// TIA Portal V16 export
// export: Created 2020-03-07T16:06:13.8131431Z, ExportSetting WithDefaults, DisplayName Totally Integrated Automation Portal, DisplayVersion V16 Update 1, DisplayName TIA Portal Version Control Interface, DisplayVersion V16, DisplayName TIA Portal Openness, DisplayVersion V16 Update 1, DisplayName STEP 7 Professional, DisplayVersion V16 Update 1, DisplayName STEP 7 Safety, DisplayVersion V16, DisplayName WinCC Professional, DisplayVersion V16 Update 1
DATA_BLOCK "function block scl_DB"   // DB3
VERSION : 0.1
// stored: AutoNumber true, DBAccessibleFromOPCUA true, InstanceOfName function block scl, InstanceOfType FB
"function block scl"
   // VAR_INPUT
   //    "a" : Int;
   //    "b" : Int;
   // END_VAR
   // VAR_OUTPUT
   //    c : Int;
   //    d : Int;
   // END_VAR
BEGIN
END_DATA_BLOCK
